FUNCTION_BLOCK FB_StationUnLoadUc_311
VAR_INPUT
	Enable:				BOOL;
	System:				REFERENCE TO ST_System;
	Station:			REFERENCE TO ST_SystemStation;
	Error:				REFERENCE TO ST_Error;
	Setting:			REFERENCE TO ST_Setting;
	Recipe:				REFERENCE TO ST_Recipe;	
	Parameter:			REFERENCE TO ST_StationUnloadUc_311;
END_VAR
VAR_OUTPUT
END_VAR
VAR
	_i:					INT;
	_arrTon:		    ARRAY[0..20] OF TON;
	_arrFbErrorTag:		ARRAY[0..20] OF FB_ErrorTag;
	_arrState:			ARRAY[0..20] OF BOOL;
	_iTakeTemp:			UINT;// 取料位
	_stHandshake: ST_StationUnloadUc_311Handshake;
END_VAR

A_Home();
A_Auto();

ACTION A_Auto:
CASE Station.iStepNow OF
	1000:
		Station.arrInfo[E_Language.Chinese]:="初始化完成 等待启动";
		IF Enable THEN
			Station.iStepNext:=1101;
		END_IF
	1101:
		Station.arrInfo[E_Language.Chinese]:="等待请求取料";
		_iTakeTemp:=0;
		IF Parameter.stHandshake.bRequestUc_L2 THEN
			_iTakeTemp:=2;
		END_IF
		IF Parameter.stHandshake.bRequestUc_L3 THEN
			_iTakeTemp:=3;
		END_IF
		IF _iTakeTemp<>0 THEN
			Station.iStepNext:=1201;
		END_IF
	1201:
		CASE _iTakeTemp OF
			2:
				IF Parameter.stHandshake.bRequestUc_L2 THEN
					Parameter.stHandshake.bResponseDismantling_Uc_L2:=TRUE;
					Station.iStepNext:=1301;
				END_IF
			3:	
				IF Parameter.stHandshake.bRequestUc_L3 THEN
					Parameter.stHandshake.bResponseDismantling_Uc_L3:=TRUE;
					Station.iStepNext:=1301;
				END_IF
		END_CASE
	1301:
		Station.arrInfo[E_Language.Chinese]:="定位至取料位";
		IF Parameter.fbAxisY.M_MoveAbs(_iTakeTemp) THEN
			Station.iStepNext:=1401;
		END_IF
	1401:
		Station.arrInfo[E_Language.Chinese]:="Z气缸下降";
		IF Parameter.fbLift.M_WorkRequest() THEN
			Station.iStepNext:=1501;
		END_IF
	1501:
		Station.arrInfo[E_Language.Chinese]:="夹紧气缸夹紧";
		IF Parameter.fbClamp.M_WorkRequest() THEN
			Station.iStepNext:=1601;
		END_IF
	1601:
		Station.arrInfo[E_Language.Chinese]:="Z气缸上升";
		IF Parameter.fbLift.M_HomeRequest() THEN
			Station.iStepNext:=1651;
		END_IF
	1651:
		Station.arrInfo[E_Language.Chinese]:="等待复位请求信号";
		CASE _iTakeTemp OF
			2:
				IF NOT Parameter.stHandshake.bRequestUc_L2 THEN
					Parameter.stHandshake.bResponseDismantling_Uc_L2:=FALSE;
					Station.iStepNext:=1901;
				END_IF
			3:	
				IF NOT Parameter.stHandshake.bRequestUc_L3 THEN
					Parameter.stHandshake.bResponseDismantling_Uc_L3:=FALSE;
					Station.iStepNext:=1901;
				END_IF
		END_CASE
	1901:
		Station.arrInfo[E_Language.Chinese]:="至下UC位";
		IF Parameter.fbAxisY.M_MoveAbs(4) THEN
			Station.iStepNext:=2001;
		END_IF
	2001:
		Station.arrInfo[E_Language.Chinese]:="Z气缸 摆动下降";
		IF Parameter.fbLift.M_WorkRequest() AND Parameter.fbSwing.M_WorkRequest() THEN
			Station.iStepNext:=2101;
		END_IF
	2101:
		Station.arrInfo[E_Language.Chinese]:="夹紧气缸松开";
		IF Parameter.fbClamp.M_HomeRequest() THEN
			Station.iStepNext:=2201;
		END_IF
	2201:
		Station.arrInfo[E_Language.Chinese]:="Z气缸 摆动上升";
		IF Parameter.fbLift.M_HomeRequest() AND Parameter.fbSwing.M_HomeRequest() THEN
			Station.iStepNext:=2301;
		END_IF
	2301:
		Station.arrInfo[E_Language.Chinese]:="至初始位";
		IF Parameter.fbAxisY.M_MoveAbs(1) THEN
			Station.iStepNext:=1101;
		END_IF
END_CASE
END_ACTION

ACTION A_Home:
CASE Station.iStepNow OF
	0:
		Station.arrInfo[E_Language.Chinese]:="等待初始化";
		Parameter.stHandshake:=_stHandshake;
		Station.iStepNext:=SEL(Enable,1000,100);
	100:
		Station.arrInfo[E_Language.Chinese]:="夹紧气缸松开";
		IF Parameter.fbClamp.M_HomeRequest() THEN
			Station.iStepNext:=200;
		END_IF
	200:
		Station.arrInfo[E_Language.Chinese]:="Z气缸上升";
		IF Parameter.fbLift.M_HomeRequest() THEN
			Station.iStepNext:=250;
		END_IF
	250:
		Station.arrInfo[E_Language.Chinese]:="摆动气缸上升";
		IF Parameter.fbSwing.M_HomeRequest() THEN
			Station.iStepNext:=300;
		END_IF
	300:
		Station.arrInfo[E_Language.Chinese]:="Y轴回零";
		IF  Parameter.fbAxisY.M_Home() THEN
			Station.iStepNext:=400;
		END_IF
	400:
		Station.arrInfo[E_Language.Chinese]:="Y轴至初始位";
		IF  Parameter.fbAxisY.M_MoveAbs(1) THEN
			Station.iStepNext:=1000;
		END_IF
END_CASE
END_ACTION

END_FUNCTION_BLOCK

(* stored: Version 1.1.0.1, ProductVersion 3.1.4024.3
   POU FB_StationUnLoadUc_311: Id {9e00e03f-db07-4f42-b955-584226488182}, SpecialFunc None
   Action A_Auto: Id {45898441-a251-4dbf-a5fc-3c03eff7716b}
   Action A_Home: Id {36e32805-0870-425b-b05c-5687922cc2c6} *)
